{attribute 'linkalways'} 
{attribute 'no_explicit_call' := 'This FB is a CLASS and must be accessed using methods or properties'}
{attribute 'enable_dynamic_creation'}
FUNCTION_BLOCK _UINT EXTENDS NumericDatatypeBase
VAR
	localData : UINT;
	activeData : REFERENCE TO UINT REF= localData;
END_VAR

PROPERTY PUBLIC Address : PVOID
GET
Address := ADR(activeData);
END_GET
END_PROPERTY

METHOD PUBLIC ClearReference
VAR_INPUT
END_VAR
activeData REF= localData;
END_METHOD

METHOD PUBLIC Clone : I_Datatype
VAR
    pClone : POINTER TO _UINT;
END_VAR
pClone := __NEW(_UINT(InitialValue := Value));
Clone := pClone^;
END_METHOD

METHOD FB_init : BOOL
VAR_INPUT
	bInitRetains : BOOL; // if TRUE, the retain variables are initialized (warm start / cold start)
	bInCopyCode : BOOL;  // if TRUE, the instance afterwards gets moved into the copy code (online change)
	InitialValue : UINT;
END_VAR
localData := InitialValue;
END_METHOD

PROPERTY PUBLIC IsFloat : BOOL
GET
IsFloat := FALSE;
END_GET
END_PROPERTY

PROPERTY PUBLIC IsSigned : BOOL
GET
IsSigned := FALSE;
END_GET
END_PROPERTY

METHOD PUBLIC MakeReferenceTo
VAR_INPUT
	ReferenceTarget : REFERENCE TO UINT;
END_VAR
activeData REF= ReferenceTarget;
END_METHOD

PROPERTY PUBLIC MaxValue : UINT
GET
MaxValue :=  DatatypeLimits.UINT_MAX_VALUE;
END_GET
END_PROPERTY

PROPERTY PUBLIC MinValue : UINT
GET
MinValue := DatatypeLimits.UINT_MIN_VALUE;
END_GET
END_PROPERTY

METHOD PROTECTED SerializeMaxValue
VAR_INPUT
	Serializer : I_Serializer;
END_VAR
Serializer.AddUint(MaxValue);
END_METHOD

METHOD PROTECTED SerializeMinValue
VAR_INPUT
	Serializer : I_Serializer;
END_VAR
Serializer.AddUint(MinValue);
END_METHOD

METHOD PUBLIC SerializeWith
VAR_INPUT
	Serializer : I_Serializer;
END_VAR
Serializer.AddUint(activeData);
END_METHOD

PROPERTY PUBLIC Size : UDINT
GET
Size := SIZEOF(activeData);
END_GET
END_PROPERTY

METHOD TryDeserializeFrom : BOOL
VAR_INPUT
	Deserializer : I_Deserializer;
	Feedback : I_DeserializerFeedback;
END_VAR
TryDeserializeFrom := Deserializer.TryGetUint(activeData, Feedback);
END_METHOD

METHOD TryMakeReferenceTo : BOOL
VAR_INPUT
	Target : I_Datatype;
END_VAR
VAR
	pTargetData : POINTER TO UINT;
END_VAR
IF NOT (Target.TypeName = TypeName) THEN
	RETURN;
END_IF

pTargetData := Target.Address;
activeData REF= pTargetData^;
TryMakeReferenceTo := TRUE;
END_METHOD

PROPERTY PUBLIC TypeName : T_MAXSTRING
GET
TypeName := 'UINT';
END_GET
END_PROPERTY

PROPERTY PUBLIC Value : REFERENCE TO UINT
GET
Value REF= activeData;
END_GET
END_PROPERTY

END_FUNCTION_BLOCK

(* stored: Version 1.1.0.1, ProductVersion 3.1.4024.12
   POU _UINT: Id {73dae905-b1b3-4651-a6d1-d1e0176f404e}, SpecialFunc None
   Folder Constructor: Id {922d2a8f-8b17-42e9-a3d2-241baf1e4522}
   Folder Protected: Id {bf20a678-ea00-461e-8ea4-457807153046}
   Property Address: Id {7b946974-e465-4392-b7ff-f57ec82ebd73}
   Get Get: Id {fde0e66f-2663-410f-b489-91d1855f7e7f}
   Method ClearReference: Id {71065f32-39af-4bb9-aa94-a92c09f2aac8}
   Method Clone: Id {227a9cfe-b1f7-41ca-9c11-d4464c5daf20}
   Method FB_init: Id {f1ba4178-7d04-41e0-aa83-6704fdc572cb}
   Property IsFloat: Id {9bc7e8a5-ffbc-4637-b9a7-eb178cf95fce}
   Get Get: Id {16e01c9f-770c-4b34-9ea8-d397d34d7daf}
   Property IsSigned: Id {d7731a3e-9f11-4760-9f11-8a1576bfdacb}
   Get Get: Id {7d87a342-b60a-4584-bb5d-fd317c7dd36f}
   Method MakeReferenceTo: Id {5b85fb77-adcc-4722-893e-3fee05ccfb5c}
   Property MaxValue: Id {ed8d0f79-f5cd-479a-a8c0-e023c76dac1e}
   Get Get: Id {b681d120-1248-42e4-929a-b16414bc6456}
   Property MinValue: Id {8b21ff72-268b-4fda-ab96-28cca7fccf6f}
   Get Get: Id {f3684f6a-fb2b-4a05-a688-05c666442a04}
   Method SerializeMaxValue: Id {dba5feb3-d4d2-4b2a-a350-561a40aab828}
   Method SerializeMinValue: Id {322efc4f-ee07-4cc1-b5ec-789b0b36c10b}
   Method SerializeWith: Id {a3cd5d92-c32d-49dc-a7f4-14e7e2f7f23c}
   Property Size: Id {553d623d-9f2e-4199-a2c3-e9310b456c89}
   Get Get: Id {ad9cf367-f7db-4e7d-ab33-527751e788a1}
   Method TryDeserializeFrom: Id {0937a836-4fc4-4775-bdd9-9a769b835e0b}
   Method TryMakeReferenceTo: Id {080c217f-a73a-4f0a-953c-d1964fa263ee}
   Property TypeName: Id {7ef2feae-632a-4f6e-a0ee-333077824a6e}
   Get Get: Id {db8030b4-e161-4e4c-a305-57fe058f3323}
   Property Value: Id {5b74dcbf-94b9-4022-bce2-2b922ffa3565}
   Get Get: Id {447582bd-79ea-424b-a79a-fe06489d2d1e} *)
